// TIA Portal V20 export
TYPE "typeSequenceControlNodeJobInterface_topTapeLoading"
// stored: Namespace Unit1.Em3
   STRUCT
      chargeJob2 : "LER_typeJobInterface";
   END_STRUCT;
END_TYPE
